// TIA Portal project "PID_2" (V16)

(* hardware
DEVICE "S71500/ET200MP-Station_1"  S7-1500 station
   slot 0: "Profilschiene_0"  Rack  6ES7 590-1***0-0AA0
   slot 1: "PLC_1"  CPU 1512C-1 PN  6ES7 512-1CK01-0AB0  V2.8
      slot 3: "CPU-Display_1"  6ES7591-1AA00-0AA0
      slot 32768: "PROFINET-Schnittstelle_1"  X1
         slot 32769: "Port_1"  X1 P1
         slot 32770: "Port_2"  X1 P2
      slot 34817: "Virtual CP interface port_1"  Virtual CP interface port  Virtual CP interface port
   slot 2: "AI 8xU/I/RTD/TC ST_1"  AI 8xU/I/RTD/TC ST  6ES7 531-7KF00-0AB0  V2.0
   slot 3: "AI 8xU/I/RTD/TC ST_2"  AI 8xU/I/RTD/TC ST  6ES7 531-7KF00-0AB0  V2.0
   slot 4: "AI 8xU/I/RTD/TC ST_3"  AI 8xU/I/RTD/TC ST  6ES7 531-7KF00-0AB0  V2.0
   slot 5: "AI 8xU/I/RTD/TC ST_4"  AI 8xU/I/RTD/TC ST  6ES7 531-7KF00-0AB0  V2.0
   slot 6: "DI 16x24VDC BA_1"  DI 16x24VDC BA  6ES7 521-1BH10-0AA0  V1.0
*)

// ===== PLC "PLC_1"  CPU 1512C-1 PN =====

VAR_GLOBAL   // PLC tag table "Standard-Variablentabelle"
   "Tag_1" AT %E0.0 : Bool;
   "Tag_2" AT %A0.0 : Bool;
   "Tag_3" AT %E0.1 : Bool;
END_VAR

VAR_GLOBAL   // PLC tag table "Inputs"
   "Flow_Rate_Sensor" AT %I0.0 : Bool;
   "Float_switch_overflow" AT %I0.1 : Bool;   // S111
   "Float_switch_threshold" AT %I0.2 : Bool;   // S112
   "Low_Level_Capacitive_Sensor" AT %I0.3 : Bool;   // B114
   "High_Level_Capacitive_Sensor" AT %I0.4 : Bool;   // B113
   "Micro_switch_valve_closed" AT %I0.5 : Bool;
   "Micro_switch_valve_open" AT %I0.6 : Bool;
   "Ultrasonic_Sensor" AT %IW96 : Int;
END_VAR

VAR_GLOBAL   // PLC tag table "Outputs"
   "Solenoid_on/off" AT %Q0.0 : Bool;
   "Heater_on/off" AT %Q0.1 : Bool;
   "Relay KF1_Pump mode" AT %Q0.2 : Bool;
   "Pump_on/off" AT %Q0.3 : Bool;
   "KF6_Proportional valve" AT %Q0.4 : Bool;
   "KF2_Fan" AT %Q0.5 : Bool;
   "Pump_P101" AT %QW96 : Int;
END_VAR

VAR_GLOBAL   // PLC tag table "Factory tags"
   "FactoryIO_running" AT %I1.3 : Bool;
   "Ultrasonic_Sensor_factory" AT %ID30 : Real;
   "Fill valve" AT %QD30 : Real;
   "Discharge valve" AT %QD34 : Real;
   "SP" AT %QD38 : DWord;
   "Flow meter" AT %ID34 : Real;
   "setpoint" AT %ID38 : Real;
   "PV" AT %QD42 : DWord;
END_VAR

// folder: Sys_par

DATA_BLOCK "parameters"   // DB2
{ S7_Optimized_Access := 'TRUE' }
VERSION : 0.1
   VAR
      "Process Value" : Real;
      setpoint : Int := 0;
      flowrate : Real;
      ModeActivate : Bool;
      ManualEnable : Bool;
      ManualValue : Real := 80.0;
      Mode : Int;
      Reset : Bool;
      float_setpoint : Real;
   END_VAR
BEGIN
END_DATA_BLOCK

// folder: (top level)

FUNCTION "height_conversion" : Void   // FC1, LAD
{ S7_Optimized_Access := 'TRUE' }
VERSION : 0.1
   VAR_INPUT
      height_sensor : Real;
      height_setpoint : Int;
   END_VAR
   VAR_OUTPUT
      scaled_height : Real;
      scaled_setpoint : Real;
   END_VAR
   VAR_TEMP
      norm_height : Real;
      norm_setpoint : Real;
   END_VAR
BEGIN

REGION Network 1: Height Conversion
   // 1. Normalize the sensor output data between 0.0 and 1.0
   // 2. Scale the normalized data between minimum and maximum scale reading
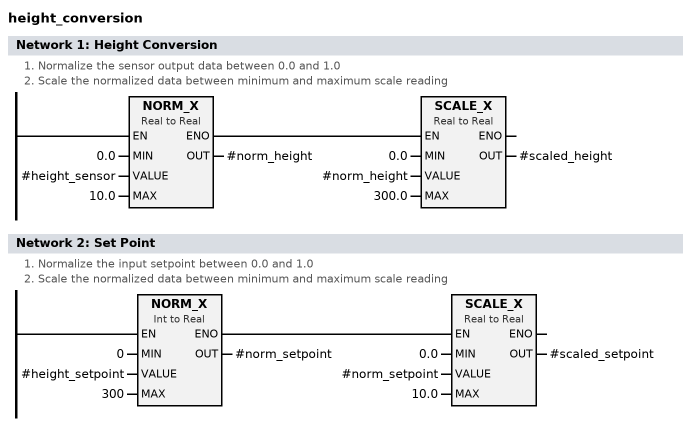
   RUNG wire#powerrail
      { S7_Templates := "[SrcType := Real, DestType := Real]" } Normalize(min := 0.0, value := #height_sensor, max := 10.0, out => #norm_height)
      { S7_Templates := "[SrcType := Real, DestType := Real]" } Scale(min := 0.0, value := #norm_height, max := 300.0, out => #scaled_height)
   END_RUNG
   // the same network as SCL:
   #norm_height := NORM_X(MIN := 0.0, VALUE := #height_sensor, MAX := 10.0);
   #scaled_height := SCALE_X(MIN := 0.0, VALUE := #norm_height, MAX := 300.0);
END_REGION

REGION Network 2: Set Point
   // 1. Normalize the input setpoint between 0.0 and 1.0
   // 2. Scale the normalized data between minimum and maximum scale reading
   RUNG wire#powerrail
      { S7_Templates := "[SrcType := Int, DestType := Real]" } Normalize(min := 0, value := #height_setpoint, max := 300, out => #norm_setpoint)
      { S7_Templates := "[SrcType := Real, DestType := Real]" } Scale(min := 0.0, value := #norm_setpoint, max := 10.0, out => #scaled_setpoint)
   END_RUNG
   // the same network as SCL:
   #norm_setpoint := NORM_X(MIN := 0, VALUE := #height_setpoint, MAX := 300);
   #scaled_setpoint := SCALE_X(MIN := 0.0, VALUE := #norm_setpoint, MAX := 10.0);
END_REGION
END_FUNCTION

FUNCTION "conversion" : Void   // FC2, LAD
{ S7_Optimized_Access := 'TRUE' }
VERSION : 0.1
   VAR_INPUT
      conv_in : Real;
   END_VAR
   VAR_OUTPUT
      conv_val : Int;
   END_VAR
   VAR_TEMP
      converted_val : Int;
   END_VAR
BEGIN

REGION Network 1
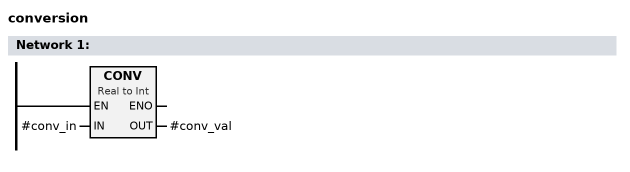
   RUNG wire#powerrail
      { S7_Templates := "[SrcType := Real, DestType := Int]" } Convert(in := #conv_in, out => #conv_val)
   END_RUNG
   // the same network as SCL:
   #conv_val := REAL_TO_INT(#conv_in);
END_REGION
END_FUNCTION

FUNCTION "MHJ-PLC-Lab-Function-S71500" : Void   // FC9000, SCL
{ S7_Optimized_Access := 'TRUE' }
VERSION : 0.1
   VAR_TEMP
      Value : Byte;
      ForCounter : Int;
   END_VAR
   VAR CONSTANT
      Value_01_DW : DWord := 16#1223_5486;
      Value_02_DW : DWord := 16#A6C9_D1F5;
   END_VAR
BEGIN

   #Value:=PEEK(area := 16#82,
        dbNumber := 0,
        byteOffset := 511);
   #Value := #Value + 1;

   POKE(area := 16#82,
        dbNumber := 0,
        byteOffset := 511,
        value := #Value);

   POKE(area := 16#82,
        dbNumber := 0,
        byteOffset := 1016,
        value := #Value_01_DW);
   POKE(area := 16#82,
        dbNumber := 0,
        byteOffset := 1020,
        value := #Value_02_DW);

   FOR #ForCounter := 0 TO 63 DO
       #Value:=PEEK(area := 16#1,
            dbNumber := 0,
            byteOffset := #ForCounter);
       POKE(area := 16#81,
            dbNumber := 0,
            byteOffset := #ForCounter,
            value := #Value);
   END_FOR;
   #Value := PEEK(area := 16#1,
                  dbNumber := 0,
                  byteOffset := 512);
   POKE(area := 16#82,
        dbNumber := 0,
        byteOffset := 512,
        value := #Value);
END_FUNCTION

ORGANIZATION_BLOCK "Main"   // OB1, LAD, ProgramCycle
TITLE = "Main Program Sweep (Cycle)"
{ S7_Optimized_Access := 'TRUE' }
VERSION : 0.1
   VAR_INPUT
      Initial_Call : Bool;   // Initial call of this OB
      Remanence : Bool;   // =True, if remanent data are available
   END_VAR
   VAR_TEMP
      setpoint_conv : Real;
   END_VAR
BEGIN

REGION Network 1
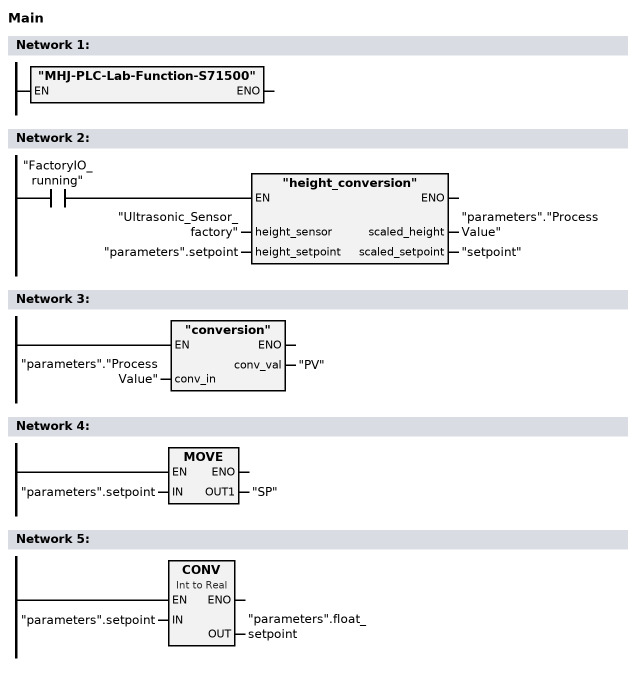
   RUNG wire#powerrail
      "MHJ-PLC-Lab-Function-S71500"()
   END_RUNG
   // the same network as SCL:
   "MHJ-PLC-Lab-Function-S71500"();
END_REGION

REGION Network 2
   RUNG wire#powerrail
      Contact( "FactoryIO_running" )
      "height_conversion"(height_sensor := "Ultrasonic_Sensor_factory", height_setpoint := "parameters".setpoint, scaled_height => "parameters"."Process Value", scaled_setpoint => "setpoint")
   END_RUNG
   // the same network as SCL:
   IF "FactoryIO_running" THEN
       "height_conversion"(height_sensor := "Ultrasonic_Sensor_factory",
                           height_setpoint := "parameters".setpoint,
                           scaled_height => "parameters"."Process Value",
                           scaled_setpoint => "setpoint");
   END_IF;
END_REGION

REGION Network 3
   RUNG wire#powerrail
      "conversion"(conv_in := "parameters"."Process Value", conv_val => "PV")
   END_RUNG
   // the same network as SCL:
   "conversion"(conv_in := "parameters"."Process Value", conv_val => "PV");
END_REGION

REGION Network 4
   RUNG wire#powerrail
      Move(in := "parameters".setpoint, out1 => "SP")
   END_RUNG
   // the same network as SCL:
   "SP" := "parameters".setpoint;
END_REGION

REGION Network 5
   RUNG wire#powerrail
      { S7_Templates := "[SrcType := Int, DestType := Real]" } Convert(in := "parameters".setpoint, out => "parameters".float_setpoint)
   END_RUNG
   // the same network as SCL:
   "parameters".float_setpoint := INT_TO_REAL("parameters".setpoint);
END_REGION
END_ORGANIZATION_BLOCK

ORGANIZATION_BLOCK "Cyclic interrupt"   // OB30, LAD, CyclicInterrupt
{ S7_Optimized_Access := 'TRUE' }
VERSION : 0.1
   VAR_INPUT
      Initial_Call : Bool;   // Initial call of this OB
      Event_Count : Int;   // Events discarded
   END_VAR
BEGIN

REGION Network 1
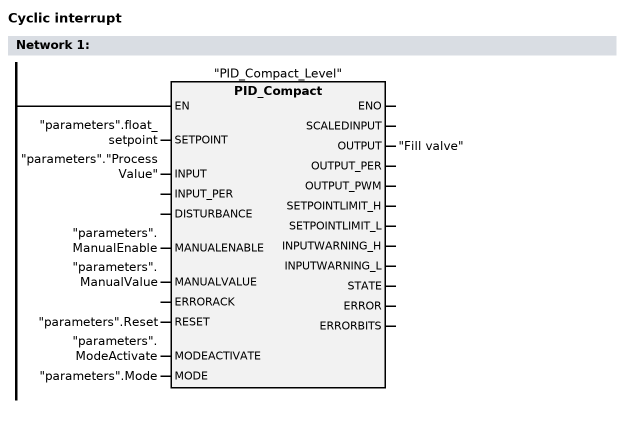
   "PID_Compact_Level"(Setpoint := "parameters".float_setpoint,   // PID_Compact
                       Input := "parameters"."Process Value",
                       ManualEnable := "parameters".ManualEnable,
                       ManualValue := "parameters".ManualValue,
                       Reset := "parameters".Reset,
                       ModeActivate := "parameters".ModeActivate,
                       Mode := "parameters".Mode,
                       Output => "Fill valve");
END_REGION
END_ORGANIZATION_BLOCK